//{attribute 'qualified_only'}
//{attribute 'strict'}
TYPE E_AI_Status  :
(
	 AI_Status_Ok,           // wszystko w normie
    AI_Status_UnderRange,   // prąd poniżej dolnego progu (np. przerwana pętla)
    AI_Status_OverRange,    // prąd powyżej górnego progu (np. zwarcie, błąd)
    AI_Status_ConfigError   // błąd konfiguracji (InMin/InMax)
);
END_TYPE

(* stored: Version 1.1.0.1, ProductVersion 3.1.4024.15
   DUT E_AI_Status: Id {1ce85c6b-a127-4910-b42c-c4beb5b48dcb} *)
